(* IEC 61131-3 sources: Codesys_MELSEC_Comm_Sample/src/SLMP_Function (part 2) *)

(* ---- FB_SlmpWriteDWordDevice.st ---- *)
FUNCTION_BLOCK FB_SlmpWriteDWordDevice
VAR_INPUT
    xExecute         : BOOL;
    sIp              : STRING;
    uiPort           : UINT;
    udiHeadDevNo     : UDINT := 0;
    uiDeviceCode     : UINT := 16#00C2; // LTN
    uiPoints         : UINT := 1; // number of 2-word points
    tTimeout         : TIME := T#2S;
    uiRetryMax       : UINT := 2;
    tReconnectDelay  : TIME := T#500MS;
    xUse4E           : BOOL := FALSE;
    xUseUdp          : BOOL := FALSE;
    uiSerialNo       : UINT := 0;
END_VAR
VAR_IN_OUT
    aWriteDWords     : ARRAY[0..SLMP_MAX_WORD_INDEX] OF UDINT;
END_VAR
VAR_OUTPUT
    xBusy            : BOOL;
    xDone            : BOOL;
    xError           : BOOL;
    diError          : DINT;
    uiRetryCount     : UINT;
    aLastResponse    : ARRAY[0..SLMP_LAST_RESPONSE_INDEX_MAX] OF BYTE;
    uiLastResponseLen: UINT;
    uiLastEndCode    : UINT;
END_VAR
VAR
    fbWriteWord      : FB_SlmpWriteWordDevice;
    aWriteWordsLocal : ARRAY[0..SLMP_MAX_WORD_INDEX] OF UINT;
    uiPointsEff      : UINT := 0;
    idx              : UINT := 0;
END_VAR

// === IMPLEMENTATION ===
uiPointsEff := uiPoints;
IF uiPointsEff > (SLMP_MAX_WORD_POINTS / 2) THEN
    uiPointsEff := SLMP_MAX_WORD_POINTS / 2;
END_IF;

FOR idx := 0 TO (uiPointsEff - 1) DO
    aWriteWordsLocal[idx * 2] := TO_UINT(aWriteDWords[idx] AND 16#0000FFFF);
    aWriteWordsLocal[idx * 2 + 1] := TO_UINT(SHR(aWriteDWords[idx], 16) AND 16#0000FFFF);
END_FOR;

fbWriteWord(
    xExecute := xExecute,
    sIp := sIp,
    uiPort := uiPort,
    udiHeadDevNo := udiHeadDevNo,
    uiDeviceCode := uiDeviceCode,
    xAutoSubCommand := FALSE,
    uiSubCommand := SLMP_SUB_WORD2,
    uiPoints := uiPointsEff,
    tTimeout := tTimeout,
    uiRetryMax := uiRetryMax,
    tReconnectDelay := tReconnectDelay,
    xUse4E := xUse4E,
    xUseUdp := xUseUdp,
    uiSerialNo := uiSerialNo,
    aWriteValues := aWriteWordsLocal
);

xBusy := fbWriteWord.xBusy;
xDone := fbWriteWord.xDone;
xError := fbWriteWord.xError;
diError := fbWriteWord.diError;
uiRetryCount := fbWriteWord.uiRetryCount;
uiLastResponseLen := fbWriteWord.uiLastResponseLen;
uiLastEndCode := fbWriteWord.uiLastEndCode;
FOR idx := 0 TO SLMP_LAST_RESPONSE_INDEX_MAX DO
    aLastResponse[idx] := fbWriteWord.aLastResponse[idx];
END_FOR;

(* ---- FB_SlmpWriteWordDevice.st ---- *)
FUNCTION_BLOCK FB_SlmpWriteWordDevice
VAR_INPUT
    xExecute         : BOOL;
    sIp              : STRING;
    uiPort           : UINT;
    udiHeadDevNo     : UDINT := 100;
    uiDeviceCode     : UINT := 16#00A8; // D
    xAutoSubCommand  : BOOL := TRUE;
    uiSubCommand     : UINT := 16#0000;
    uiPoints         : UINT := 1;
    tTimeout         : TIME := T#2S;
    uiRetryMax       : UINT := 2;
    tReconnectDelay  : TIME := T#500MS;
    xUse4E           : BOOL := FALSE;
    xUseUdp          : BOOL := FALSE;
    uiSerialNo       : UINT := 0;
END_VAR
VAR_IN_OUT
    aWriteValues     : ARRAY[0..SLMP_MAX_WORD_INDEX] OF UINT;
END_VAR
VAR_OUTPUT
    xBusy            : BOOL;
    xDone            : BOOL;
    xError           : BOOL;
    diError          : DINT;
    uiRetryCount     : UINT;
    aLastResponse    : ARRAY[0..SLMP_LAST_RESPONSE_INDEX_MAX] OF BYTE;
    uiLastResponseLen: UINT;
    uiLastEndCode    : UINT;
END_VAR
VAR
    step             : INT := 0;
    xExecPrev        : BOOL := FALSE;

    fbCore           : FB_SlmpCore;

    tx               : ARRAY[0..SLMP_WRITE_TX_INDEX_MAX] OF BYTE;
    rx               : ARRAY[0..SLMP_LAST_RESPONSE_INDEX_MAX] OF BYTE;
    txLen            : LINT := 0;
    rxLen            : LINT := 0;
    lenReq           : UINT := 0;
    endCode          : UINT := 0;

    uiPointsReq      : UINT := 0;
    uiPointsEff      : UINT := 0;
    uiPointsProto    : UINT := 0;
    uiSubCmdEff      : UINT := 0;
    xWord2Mode       : BOOL := FALSE;
    idx              : UINT := 0;
    aWriteValuesLocal: ARRAY[0..SLMP_MAX_WORD_INDEX] OF UINT;
    iDataStart       : DINT := 21;
    iEndCodeStart    : DINT := 9;
    iMinRxLen        : LINT := 11;
    uiRxSerialNo     : UINT := 0;
    uiCopyLen        : UINT := 0;
    iPayloadBytes    : LINT := 0;

    xStateTimeout    : BOOL := FALSE;
    xRetryTiming     : BOOL := FALSE;
    fbTimeout        : TON;
    fbReconnect      : TON;
END_VAR

// === IMPLEMENTATION ===
IF (xExecute AND NOT xExecPrev) THEN
    xBusy := TRUE;
    xDone := FALSE;
    xError := FALSE;
    diError := 0;
    uiRetryCount := 0;
    uiLastResponseLen := 0;
    uiLastEndCode := 0;
    FOR idx := 0 TO SLMP_LAST_RESPONSE_INDEX_MAX DO
        aLastResponse[idx] := 0;
    END_FOR;
    step := 10;
END_IF;
xExecPrev := xExecute;

xStateTimeout := (step = 20) OR (step = 40) OR (step = 50);
fbTimeout(IN := xStateTimeout, PT := tTimeout);
fbReconnect(IN := xRetryTiming, PT := tReconnectDelay);

IF (step <> 0) AND (step <> 80) AND fbTimeout.Q THEN
    diError := -2010;
    xError := TRUE;
    step := 90;
END_IF;

CASE step OF
    0:
        xRetryTiming := FALSE;

    10:
        uiSubCmdEff := F_SlmpResolveSubCommand(
            uiDeviceCode := uiDeviceCode,
            xAutoSubCommand := xAutoSubCommand,
            uiSubCommand := uiSubCommand
        );
        xWord2Mode := (uiSubCmdEff = SLMP_SUB_WORD2);

        uiPointsReq := uiPoints;
        IF uiPointsReq = 0 THEN
            diError := -2000;
            xError := TRUE;
            xBusy := FALSE;
            step := 0;
        ELSE
            uiPointsEff := F_SlmpClampPoints(uiPoints := uiPointsReq, xBitMode := FALSE);
            IF xWord2Mode THEN
                IF uiPointsEff > (SLMP_MAX_WORD_POINTS / 2) THEN
                    uiPointsEff := SLMP_MAX_WORD_POINTS / 2;
                END_IF;
                uiPointsProto := uiPointsEff * 2;
            ELSE
                uiPointsProto := uiPointsEff;
            END_IF;
        END_IF;

        FOR idx := 0 TO SLMP_MAX_WORD_INDEX DO
            aWriteValuesLocal[idx] := aWriteValues[idx];
        END_FOR;

        IF NOT xError THEN
            step := 20;
        END_IF;

    20:
        IF fbCore.OpenAndConnect(sIp := sIp, uiPort := uiPort, xUseUdp := xUseUdp) THEN
            step := 30;
        ELSE
            CASE fbCore.diLastError OF
                -1: diError := -2001;
                -2: diError := -2005;
                -3: diError := -2002;
            ELSE
                diError := -2002;
            END_CASE;
            xError := TRUE;
            step := 90;
        END_IF;

    30:
        IF xUse4E THEN
            iDataStart := 25;
            iEndCodeStart := 13;
            iMinRxLen := 15;
        ELSE
            iDataStart := 21;
            iEndCodeStart := 9;
            iMinRxLen := 11;
        END_IF;

        IF xWord2Mode THEN
            iPayloadBytes := TO_LINT(uiPointsEff) * 4;
        ELSE
            iPayloadBytes := TO_LINT(uiPointsEff) * 2;
        END_IF;
        lenReq := TO_UINT(12 + TO_UINT(iPayloadBytes));

        IF xUse4E THEN
            tx[0] := 16#54; tx[1] := 16#00;
            tx[2] := TO_BYTE(uiSerialNo AND 16#00FF);
            tx[3] := TO_BYTE(SHR(uiSerialNo, 8) AND 16#00FF);
            tx[4] := 16#00; tx[5] := 16#00;
            tx[6] := 16#00;
            tx[7] := 16#FF;
            tx[8] := 16#FF; tx[9] := 16#03;
            tx[10] := 16#00;
            tx[11] := TO_BYTE(lenReq AND 16#00FF);
            tx[12] := TO_BYTE(SHR(lenReq, 8) AND 16#00FF);
            tx[13] := 16#10; tx[14] := 16#00;
            tx[15] := 16#01; tx[16] := 16#14;
            tx[17] := TO_BYTE(uiSubCmdEff AND 16#00FF);
            tx[18] := TO_BYTE(SHR(uiSubCmdEff, 8) AND 16#00FF);
            tx[19] := TO_BYTE(udiHeadDevNo AND 16#000000FF);
            tx[20] := TO_BYTE(SHR(udiHeadDevNo, 8) AND 16#000000FF);
            tx[21] := TO_BYTE(SHR(udiHeadDevNo, 16) AND 16#000000FF);
            tx[22] := TO_BYTE(uiDeviceCode AND 16#00FF);
            tx[23] := TO_BYTE(uiPointsProto AND 16#00FF);
            tx[24] := TO_BYTE(SHR(uiPointsProto, 8) AND 16#00FF);
        ELSE
            tx[0] := 16#50; tx[1] := 16#00;
            tx[2] := 16#00;
            tx[3] := 16#FF;
            tx[4] := 16#FF; tx[5] := 16#03;
            tx[6] := 16#00;
            tx[7] := TO_BYTE(lenReq AND 16#00FF);
            tx[8] := TO_BYTE(SHR(lenReq, 8) AND 16#00FF);
            tx[9] := 16#10; tx[10] := 16#00;
            tx[11] := 16#01; tx[12] := 16#14;
            tx[13] := TO_BYTE(uiSubCmdEff AND 16#00FF);
            tx[14] := TO_BYTE(SHR(uiSubCmdEff, 8) AND 16#00FF);
            tx[15] := TO_BYTE(udiHeadDevNo AND 16#000000FF);
            tx[16] := TO_BYTE(SHR(udiHeadDevNo, 8) AND 16#000000FF);
            tx[17] := TO_BYTE(SHR(udiHeadDevNo, 16) AND 16#000000FF);
            tx[18] := TO_BYTE(uiDeviceCode AND 16#00FF);
            tx[19] := TO_BYTE(uiPointsProto AND 16#00FF);
            tx[20] := TO_BYTE(SHR(uiPointsProto, 8) AND 16#00FF);
        END_IF;

        IF xWord2Mode THEN
            FOR idx := 0 TO (uiPointsEff - 1) DO
                tx[iDataStart + TO_DINT(idx) * 4] := TO_BYTE(aWriteValuesLocal[idx * 2] AND 16#00FF);
                tx[iDataStart + TO_DINT(idx) * 4 + 1] := TO_BYTE(SHR(aWriteValuesLocal[idx * 2], 8) AND 16#00FF);
                tx[iDataStart + TO_DINT(idx) * 4 + 2] := TO_BYTE(aWriteValuesLocal[idx * 2 + 1] AND 16#00FF);
                tx[iDataStart + TO_DINT(idx) * 4 + 3] := TO_BYTE(SHR(aWriteValuesLocal[idx * 2 + 1], 8) AND 16#00FF);
            END_FOR;
        ELSE
            FOR idx := 0 TO (uiPointsEff - 1) DO
                tx[iDataStart + TO_DINT(idx) * 2] := TO_BYTE(aWriteValuesLocal[idx] AND 16#00FF);
                tx[iDataStart + TO_DINT(idx) * 2 + 1] := TO_BYTE(SHR(aWriteValuesLocal[idx], 8) AND 16#00FF);
            END_FOR;
        END_IF;

        txLen := TO_LINT(iDataStart) + iPayloadBytes;
        step := 40;

    40:
        IF NOT fbCore.SendBytes(pData := ADR(tx[0]), liLen := txLen) THEN
            diError := -2003;
            xError := TRUE;
            step := 90;
        ELSE
            step := 50;
        END_IF;

    50:
        rxLen := fbCore.RecvBytes(pData := ADR(rx[0]), liMaxLen := SIZEOF(rx));
        IF rxLen > 0 THEN
            uiCopyLen := 0;
            IF rxLen > TO_LINT(SLMP_LAST_RESPONSE_INDEX_MAX + 1) THEN
                uiCopyLen := SLMP_LAST_RESPONSE_INDEX_MAX + 1;
            ELSE
                uiCopyLen := TO_UINT(rxLen);
            END_IF;
            uiLastResponseLen := uiCopyLen;
            IF uiCopyLen > 0 THEN
                FOR idx := 0 TO (uiCopyLen - 1) DO
                    aLastResponse[idx] := rx[idx];
                END_FOR;
            END_IF;
            IF rxLen < iMinRxLen THEN
                diError := -2004;
                xError := TRUE;
                step := 90;
            ELSE
                IF xUse4E THEN
                    uiRxSerialNo := TO_UINT(rx[2]) OR SHL(TO_UINT(rx[3]), 8);
                    IF uiRxSerialNo <> uiSerialNo THEN
                        // Drop stale frame and keep waiting until timeout.
                        rxLen := 0;
                        uiLastResponseLen := 0;
                    END_IF;
                END_IF;
            END_IF;
            IF (NOT xError) AND (rxLen > 0) THEN
                endCode := TO_UINT(rx[iEndCodeStart]) OR SHL(TO_UINT(rx[iEndCodeStart + 1]), 8);
                uiLastEndCode := endCode;
                IF endCode <> 0 THEN
                    diError := TO_DINT(endCode);
                    xError := TRUE;
                    step := 90;
                ELSE
                    xDone := TRUE;
                    xBusy := FALSE;
                    step := 90;
                END_IF;
            END_IF;
        END_IF;

    80:
        xRetryTiming := TRUE;
        IF fbReconnect.Q THEN
            xRetryTiming := FALSE;
            step := 10;
        END_IF;

    90:
        IF xError THEN
            fbCore.CloseSocket();
        END_IF;

        IF xError AND (uiRetryCount < uiRetryMax) THEN
            uiRetryCount := uiRetryCount + 1;
            xError := FALSE;
            step := 80;
        ELSE
            xBusy := FALSE;
            step := 0;
        END_IF;
END_CASE;

(* ---- FB_SlmpWriteWordService.st ---- *)
FUNCTION_BLOCK FB_SlmpWriteWordService
VAR_INPUT
    xExecute        : BOOL;
    sIp             : STRING;
    uiPort          : UINT;
    udiHeadDevNo    : UDINT;
    uiDeviceCode    : UINT;
    uiPoints        : UINT;
    tTimeout        : TIME := T#2S;
    uiRetryMax      : UINT := 2;
    tReconnectDelay : TIME := T#500MS;
    xUse4E          : BOOL := FALSE;
    xUseUdp         : BOOL := FALSE;
    uiSerialNo      : UINT := 1;
END_VAR
VAR_IN_OUT
    aWriteValues    : ARRAY[0..SLMP_MAX_WORD_INDEX] OF UINT;
END_VAR
VAR_OUTPUT
    xBusy           : BOOL;
    xDone           : BOOL;
    xError          : BOOL;
    diError         : DINT;
    uiRetryCount    : UINT;
    aLastResponse   : ARRAY[0..SLMP_LAST_RESPONSE_INDEX_MAX] OF BYTE;
    uiLastResponseLen : UINT;
    uiLastEndCode   : UINT;
END_VAR
VAR
    fbWriteWord     : FB_SlmpWriteWordDevice;
    udInstanceId    : UDINT := 0;

    xExecPrev       : BOOL := FALSE;
    xPending        : BOOL := FALSE;
    xActive         : BOOL := FALSE;
    xExecPulse      : BOOL := FALSE;
    iLockIdx        : INT := -1;

    udiHeadLatched  : UDINT := 0;
    uiDeviceLatched : UINT := 0;
    uiPointsLatched : UINT := 0;
    uiSerialActive  : UINT := 0;
    aWriteLatched   : ARRAY[0..SLMP_MAX_WORD_INDEX] OF UINT;

    idx             : UINT;
    uiSerialEff     : UINT;
    iSlot           : INT;
    iFreeSlot       : INT;
    xLocked         : BOOL;
END_VAR

// === IMPLEMENTATION ===
IF udInstanceId = 0 THEN
    GVL_SlmpRuntime.g_udServiceInstanceCounter := GVL_SlmpRuntime.g_udServiceInstanceCounter + 1;
    udInstanceId := GVL_SlmpRuntime.g_udServiceInstanceCounter;
    IF udInstanceId = 0 THEN
        udInstanceId := 1;
    END_IF;
END_IF;

IF xExecute AND (NOT xExecPrev) THEN
    IF (NOT xPending) AND (NOT xActive) THEN
        udiHeadLatched := udiHeadDevNo;
        uiDeviceLatched := uiDeviceCode;
        uiPointsLatched := uiPoints;
        FOR idx := 0 TO SLMP_MAX_WORD_INDEX DO
            aWriteLatched[idx] := aWriteValues[idx];
        END_FOR;
        xDone := FALSE;
        xError := FALSE;
        diError := 0;
        uiRetryCount := 0;
        xPending := TRUE;
    END_IF;
END_IF;
xExecPrev := xExecute;

xExecPulse := FALSE;
IF xPending AND (NOT xActive) THEN
    xLocked := FALSE;
    iFreeSlot := -1;
    FOR iSlot := 0 TO 7 DO
        IF (GVL_SlmpRuntime.g_aLockOwner[iSlot] <> 0) AND
           (GVL_SlmpRuntime.g_aLockIp[iSlot] = sIp) AND
           (GVL_SlmpRuntime.g_aLockPort[iSlot] = uiPort) AND
           (GVL_SlmpRuntime.g_aLockUseUdp[iSlot] = xUseUdp) THEN
            xLocked := TRUE;
            EXIT;
        END_IF;
        IF (iFreeSlot < 0) AND (GVL_SlmpRuntime.g_aLockOwner[iSlot] = 0) THEN
            iFreeSlot := iSlot;
        END_IF;
    END_FOR;

    IF (NOT xLocked) AND (iFreeSlot >= 0) THEN
        GVL_SlmpRuntime.g_aLockOwner[iFreeSlot] := udInstanceId;
        GVL_SlmpRuntime.g_aLockIp[iFreeSlot] := sIp;
        GVL_SlmpRuntime.g_aLockPort[iFreeSlot] := uiPort;
        GVL_SlmpRuntime.g_aLockUseUdp[iFreeSlot] := xUseUdp;
        iLockIdx := iFreeSlot;

        xActive := TRUE;
        xExecPulse := TRUE;
        IF xUse4E THEN
            uiSerialActive := F_SlmpNextSerialNo(uiSeed := uiSerialNo);
        END_IF;
    END_IF;
END_IF;

IF xActive THEN
    IF xUse4E THEN
        uiSerialEff := uiSerialActive;
        IF uiSerialEff = 0 THEN
            uiSerialEff := 1;
        END_IF;
    ELSE
        uiSerialEff := uiSerialNo;
    END_IF;

    fbWriteWord(
        xExecute := xExecPulse,
        sIp := sIp,
        uiPort := uiPort,
        udiHeadDevNo := udiHeadLatched,
        uiDeviceCode := uiDeviceLatched,
        xAutoSubCommand := TRUE,
        uiSubCommand := 0,
        uiPoints := uiPointsLatched,
        tTimeout := tTimeout,
        uiRetryMax := uiRetryMax,
        tReconnectDelay := tReconnectDelay,
        xUse4E := xUse4E,
        xUseUdp := xUseUdp,
        uiSerialNo := uiSerialEff,
        aWriteValues := aWriteLatched
    );
ELSE
    xBusy := xPending;
    IF NOT xExecute THEN
        xDone := FALSE;
        xError := FALSE;
        diError := 0;
        uiRetryCount := 0;
    END_IF;
    RETURN;
END_IF;

xBusy := fbWriteWord.xBusy;
xDone := fbWriteWord.xDone;
xError := fbWriteWord.xError;
diError := fbWriteWord.diError;
uiRetryCount := fbWriteWord.uiRetryCount;
FOR idx := 0 TO SLMP_LAST_RESPONSE_INDEX_MAX DO
    aLastResponse[idx] := fbWriteWord.aLastResponse[idx];
END_FOR;
uiLastResponseLen := fbWriteWord.uiLastResponseLen;
uiLastEndCode := fbWriteWord.uiLastEndCode;

IF fbWriteWord.xDone OR fbWriteWord.xError THEN
    xPending := FALSE;
    xActive := FALSE;
    IF iLockIdx >= 0 THEN
        GVL_SlmpRuntime.g_aLockOwner[iLockIdx] := 0;
        GVL_SlmpRuntime.g_aLockIp[iLockIdx] := '';
        GVL_SlmpRuntime.g_aLockPort[iLockIdx] := 0;
        GVL_SlmpRuntime.g_aLockUseUdp[iLockIdx] := FALSE;
        iLockIdx := -1;
    END_IF;
END_IF;

(* ---- FB_SlmpCore.CloseSocket.st ---- *)
METHOD CloseSocket

// === IMPLEMENTATION ===

IF iSockSlot < 0 THEN
    RETURN;
END_IF;

IF GVL_SlmpRuntime.g_aSockHandle[iSockSlot] <> RTS_INVALID_HANDLE THEN
    SysSockClose(GVL_SlmpRuntime.g_aSockHandle[iSockSlot]);
    GVL_SlmpRuntime.g_aSockHandle[iSockSlot] := RTS_INVALID_HANDLE;
END_IF;
GVL_SlmpRuntime.g_aSockConnected[iSockSlot] := FALSE;
GVL_SlmpRuntime.g_aSockIp[iSockSlot] := '';
GVL_SlmpRuntime.g_aSockPort[iSockSlot] := 0;
GVL_SlmpRuntime.g_aSockUseUdp[iSockSlot] := FALSE;
iSockSlot := -1;

(* ---- FB_SlmpCore.OpenAndConnect.st ---- *)
METHOD OpenAndConnect : BOOL
VAR_INPUT
    sIp    : STRING;
    uiPort : UINT;
    xUseUdp : BOOL := FALSE;
END_VAR
VAR
    iSlot  : INT;
    iFree  : INT;
END_VAR

// === IMPLEMENTATION ===
OpenAndConnect := FALSE;
diLastError := 0;

// Reuse already bound and connected slot for same destination.
IF iSockSlot >= 0 THEN
    IF GVL_SlmpRuntime.g_aSockConnected[iSockSlot] AND
       (GVL_SlmpRuntime.g_aSockIp[iSockSlot] = sIp) AND
       (GVL_SlmpRuntime.g_aSockPort[iSockSlot] = uiPort) AND
       (GVL_SlmpRuntime.g_aSockUseUdp[iSockSlot] = xUseUdp) THEN
        OpenAndConnect := TRUE;
        RETURN;
    END_IF;
    iSockSlot := -1;
END_IF;

// Find existing connected slot for destination, or a free slot.
iFree := -1;
FOR iSlot := 0 TO 7 DO
    IF GVL_SlmpRuntime.g_aSockConnected[iSlot] AND
       (GVL_SlmpRuntime.g_aSockIp[iSlot] = sIp) AND
       (GVL_SlmpRuntime.g_aSockPort[iSlot] = uiPort) AND
       (GVL_SlmpRuntime.g_aSockUseUdp[iSlot] = xUseUdp) THEN
        iSockSlot := iSlot;
        OpenAndConnect := TRUE;
        RETURN;
    END_IF;

    IF (iFree < 0) AND (NOT GVL_SlmpRuntime.g_aSockConnected[iSlot]) THEN
        iFree := iSlot;
    END_IF;
END_FOR;

IF iFree < 0 THEN
    diLastError := -6; // no free shared socket slot
    RETURN;
END_IF;

IF xUseUdp THEN
    GVL_SlmpRuntime.g_aSockHandle[iFree] := SysSockCreate(SOCKET_AF_INET, SOCKET_DGRAM, SOCKET_IPPROTO_UDP, ADR(res));
ELSE
    GVL_SlmpRuntime.g_aSockHandle[iFree] := SysSockCreate(SOCKET_AF_INET, SOCKET_STREAM, SOCKET_IPPROTO_IP, ADR(res));
END_IF;
IF GVL_SlmpRuntime.g_aSockHandle[iFree] = RTS_INVALID_HANDLE THEN
    diLastError := -1;
    RETURN;
END_IF;

liRet := SysSockInetAddr(sIp, ADR(ipAddr));
IF liRet <> 0 THEN
    diLastError := -2;
    SysSockClose(GVL_SlmpRuntime.g_aSockHandle[iFree]);
    GVL_SlmpRuntime.g_aSockHandle[iFree] := RTS_INVALID_HANDLE;
    RETURN;
END_IF;

sa.sin_family := SOCKET_AF_INET;
sa.sin_port := SysSockHtons(uiPort);
sa.sin_addr := ipAddr;

liRet := SysSockConnect(GVL_SlmpRuntime.g_aSockHandle[iFree], ADR(sa), SIZEOF(sa));
IF liRet <> 0 THEN
    diLastError := -3;
    SysSockClose(GVL_SlmpRuntime.g_aSockHandle[iFree]);
    GVL_SlmpRuntime.g_aSockHandle[iFree] := RTS_INVALID_HANDLE;
    RETURN;
END_IF;

GVL_SlmpRuntime.g_aSockConnected[iFree] := TRUE;
GVL_SlmpRuntime.g_aSockIp[iFree] := sIp;
GVL_SlmpRuntime.g_aSockPort[iFree] := uiPort;
GVL_SlmpRuntime.g_aSockUseUdp[iFree] := xUseUdp;
iSockSlot := iFree;
OpenAndConnect := TRUE;

(* ---- FB_SlmpCore.RecvBytes.st ---- *)
METHOD RecvBytes : LINT
VAR_INPUT
    pData    : POINTER TO BYTE;
    liMaxLen : LINT;
END_VAR
VAR
    fdRead   : SOCKET_FD_SET;
    tv       : SOCKET_TIMEVAL;
    diReady  : DINT := 0;
    rtResult : RTS_IEC_RESULT := 0;
END_VAR

// === IMPLEMENTATION ===
diLastError := 0;
IF iSockSlot < 0 THEN
    diLastError := -5;
    RecvBytes := 0;
    RETURN;
END_IF;

// Avoid blocking task: recv only when socket is readable.
rtResult := SysSockFdZero(fdRead);
rtResult := SysSockFdInit(GVL_SlmpRuntime.g_aSockHandle[iSockSlot], fdRead);
tv.tv_sec := 0;
tv.tv_usec := 0;
diReady := 0;
rtResult := SysSockSelect(
    SOCKET_FD_SETSIZE,
    ADR(fdRead),
    0,
    0,
    ADR(tv),
    ADR(diReady)
);
IF (rtResult <> 0) OR (diReady <= 0) THEN
    RecvBytes := 0;
    RETURN;
END_IF;

RecvBytes := SysSockRecv(GVL_SlmpRuntime.g_aSockHandle[iSockSlot], pData, liMaxLen, 0, ADR(res));
IF RecvBytes <= 0 THEN
    diLastError := -5;
    RecvBytes := 0;
END_IF;

(* ---- FB_SlmpCore.SendBytes.st ---- *)
METHOD SendBytes : BOOL
VAR_INPUT
    pData : POINTER TO BYTE;
    liLen : LINT;
END_VAR
VAR
    uiCopyLen : UINT := 0;
    idx       : UINT := 0;
END_VAR

// === IMPLEMENTATION ===
SendBytes := FALSE;
diLastError := 0;

IF iSockSlot < 0 THEN
    diLastError := -4;
    RETURN;
END_IF;

GVL_SlmpRuntime.g_iLastTxSockSlot := iSockSlot;
GVL_SlmpRuntime.g_uiLastTxLen := 0;
IF liLen > 0 THEN
    IF liLen > TO_LINT(SLMP_WRITE_TX_INDEX_MAX + 1) THEN
        uiCopyLen := SLMP_WRITE_TX_INDEX_MAX + 1;
    ELSE
        uiCopyLen := TO_UINT(liLen);
    END_IF;
    GVL_SlmpRuntime.g_uiLastTxLen := uiCopyLen;
    FOR idx := 0 TO (uiCopyLen - 1) DO
        GVL_SlmpRuntime.g_aLastTx[idx] := pData[idx];
    END_FOR;
END_IF;

liRet := SysSockSend(GVL_SlmpRuntime.g_aSockHandle[iSockSlot], pData, liLen, 0, ADR(res));
IF liRet <= 0 THEN
    diLastError := -4;
    CloseSocket();
    RETURN;
END_IF;

SendBytes := TRUE;

(* ---- FB_SlmpReadDevice.CalcNeedRxLen.st ---- *)
METHOD CalcNeedRxLen : LINT

// === IMPLEMENTATION ===

IF xBitMode THEN
    CalcNeedRxLen := iDataStart + TO_LINT((uiPointsEff + 1) / 2);
ELSE
    CalcNeedRxLen := iDataStart + TO_LINT(uiPointsEff) * 2;
END_IF;

(* ---- FB_SlmpReadDevice.DecodeBitArray.st ---- *)
METHOD DecodeBitArray : BOOL

// === IMPLEMENTATION ===

DecodeBitArray := TRUE;

FOR idx := 0 TO (uiPointsEff - 1) DO
    iByteOffset := iDataStart + TO_DINT(idx / 2);
    byData := rx[iByteOffset];
    IF (idx MOD 2) = 0 THEN
        aBits[idx] := (byData AND 16#F0) <> 0;
    ELSE
        aBits[idx] := (byData AND 16#0F) <> 0;
    END_IF;
    IF idx <= SLMP_MAX_WORD_INDEX THEN
        IF aBits[idx] THEN
            aValues[idx] := 1;
        ELSE
            aValues[idx] := 0;
        END_IF;
    END_IF;
END_FOR;

uiReadBits := uiPointsEff;
uiReadWords := 0;

IF uiPointsEff > 0 THEN
    IF aBits[0] THEN
        uiValue0 := 1;
    ELSE
        uiValue0 := 0;
    END_IF;
END_IF;

(* ---- FB_SlmpReadDevice.DecodeReadData.st ---- *)
METHOD DecodeReadData : BOOL

// === IMPLEMENTATION ===

DecodeReadData := TRUE;

IF xBitMode THEN
    DecodeReadData := DecodeBitArray();
ELSE
    DecodeReadData := DecodeWordArray();
END_IF;

(* ---- FB_SlmpReadDevice.DecodeWordArray.st ---- *)
METHOD DecodeWordArray : BOOL

// === IMPLEMENTATION ===

DecodeWordArray := TRUE;

FOR idx := 0 TO (uiPointsEff - 1) DO
    aValues[idx] := TO_UINT(rx[iDataStart + TO_DINT(idx) * 2]) OR SHL(TO_UINT(rx[iDataStart + TO_DINT(idx) * 2 + 1]), 8);
END_FOR;

uiReadWords := uiPointsEff;
uiReadBits := 0;
uiValue0 := aValues[0];

(* ---- FB_SlmpWriteDevice.BuildBitPayload.st ---- *)
METHOD BuildBitPayload : LINT

// === IMPLEMENTATION ===

BuildBitPayload := TO_LINT((uiPointsEff + 1) / 2);

FOR idx := 0 TO ((uiPointsEff - 1) / 2) DO
    tx[iDataStart + TO_DINT(idx)] := 16#00;
END_FOR;

FOR idx := 0 TO (uiPointsEff - 1) DO
    iByteOffset := iDataStart + TO_DINT(idx / 2);
    IF aWriteBits[idx] THEN
        IF (idx MOD 2) = 0 THEN
            tx[iByteOffset] := TO_BYTE(tx[iByteOffset] OR 16#10);
        ELSE
            tx[iByteOffset] := TO_BYTE(tx[iByteOffset] OR 16#01);
        END_IF;
    END_IF;
END_FOR;

(* ---- FB_SlmpWriteDevice.BuildWordPayload.st ---- *)
METHOD BuildWordPayload : LINT

// === IMPLEMENTATION ===

BuildWordPayload := TO_LINT(uiPointsEff) * 2;

FOR idx := 0 TO (uiPointsEff - 1) DO
    tx[iDataStart + TO_DINT(idx) * 2] := TO_BYTE(aWriteValuesLocal[idx] AND 16#00FF);
    tx[iDataStart + TO_DINT(idx) * 2 + 1] := TO_BYTE(SHR(aWriteValuesLocal[idx], 8) AND 16#00FF);
END_FOR;

(* ---- FB_SlmpWriteDevice.BuildWritePayload.st ---- *)
METHOD BuildWritePayload : LINT

// === IMPLEMENTATION ===

IF xBitMode THEN
    BuildWritePayload := BuildBitPayload();
ELSE
    BuildWritePayload := BuildWordPayload();
END_IF;
